  MoveL 9057 to (-391.21, -17.4, -14.38) mm, rotated rx 180 ry 0 rz 0.01 deg; joints [25.24, -41.819, 95.967, -150.014, 58.606, 164.358]
  MoveL 9058 to (-397.59, -19.12, -14.63) mm, rotated rx -180 ry 0 rz 0.01 deg; joints [25.086, -41.563, 95.461, -150.11, 58.344, 164.303]
  MoveL 9059 to (-398.57, -25.65, -14.87) mm, rotated rx 180 ry 0 rz 0.01 deg; joints [24.857, -41.636, 95.647, -150.402, 58.376, 164.507]
  MoveL 9060 to (-392.98, -29.17, -15.11) mm, rotated rx 180 ry 0 rz 0.01 deg; joints [24.827, -41.935, 96.3, -150.543, 58.676, 164.73]
  MoveL 9061 to (-387.52, -25.46, -15.36) mm, rotated rx 180 ry 0 rz 0.01 deg; joints [25.033, -42.088, 96.637, -150.367, 58.894, 164.714]
  MoveL 9062 to (-388.73, -18.96, -15.6) mm, rotated rx 180 ry 0 rz 0.01 deg; joints [25.228, -41.898, 96.253, -150.09, 58.782, 164.486]
  MoveL 9063 to (-395.17, -17.47, -15.85) mm, rotated rx -180 ry 0 rz 0.01 deg; joints [25.178, -41.578, 95.607, -150.047, 58.485, 164.325]
  MoveL 9064 to (-399.11, -22.77, -16.09) mm, rotated rx 180 ry 0 rz 0.01 deg; joints [24.944, -41.498, 95.473, -150.293, 58.37, 164.434]
  MoveL 9065 to (-395.84, -28.51, -16.33) mm, rotated rx 180 ry 0 rz 0.01 deg; joints [24.806, -41.739, 96.011, -150.538, 58.588, 164.688]
  MoveL 9066 to (-389.27, -27.81, -16.58) mm, rotated rx -180 ry 0 rz 0.01 deg; joints [24.93, -41.998, 96.574, -150.49, 58.888, 164.79]
  MoveL 9067 to (-387.28, -21.51, -16.82) mm, rotated rx 180 ry 0 rz 0.01 deg; joints [25.168, -41.951, 96.488, -150.212, 58.922, 164.627]
  MoveL 9068 to (-392.25, -17.16, -17.07) mm, rotated rx -180 ry 0 rz 0.01 deg; joints [25.234, -41.64, 95.854, -150.041, 58.661, 164.4]
  MoveL 9069 to (-398.23, -19.98, -17.31) mm, rotated rx 180 ry 0 rz 0.01 deg; joints [25.05, -41.424, 95.431, -150.184, 58.429, 164.389]
  MoveL 9070 to (-398.04, -26.58, -17.55) mm, rotated rx 180 ry 0 rz 0.01 deg; joints [24.837, -41.548, 95.725, -150.475, 58.515, 164.616]
  MoveL 9071 to (-391.92, -29.05, -17.8) mm, rotated rx -180 ry 0 rz 0.01 deg; joints [24.849, -41.849, 96.383, -150.569, 58.829, 164.814]
  MoveL 9072 to (-387.2, -24.44, -18.04) mm, rotated rx 180 ry 0 rz 0.01 deg; joints [25.073, -41.952, 96.614, -150.355, 59.004, 164.755]
  MoveL 9073 to (-389.54, -18.26, -18.29) mm, rotated rx -180 ry 0 rz 0.01 deg; joints [25.241, -41.72, 96.142, -150.096, 58.844, 164.518]
  MoveL 9074 to (-396.13, -17.93, -18.53) mm, rotated rx 180 ry 0 rz 0.01 deg; joints [25.15, -41.417, 95.53, -150.104, 58.55, 164.392]
  MoveL 9075 to (-399.08, -23.84, -18.77) mm, rotated rx -180 ry 0 rz 0.01 deg; joints [24.912, -41.391, 95.512, -150.374, 58.487, 164.538]
  MoveL 9076 to (-394.85, -28.91, -19.02) mm, rotated rx 180 ry 0 rz 0.01 deg; joints [24.81, -41.661, 96.108, -150.587, 58.742, 164.787]
  MoveL 9077 to (-388.51, -27.06, -19.26) mm, rotated rx 180 ry 0 rz 0.01 deg; joints [24.968, -41.887, 96.602, -150.489, 59.02, 164.848]
  MoveL 9078 to (-387.66, -20.51, -19.51) mm, rotated rx -180 ry 0 rz 0.01 deg; joints [25.197, -41.786, 96.402, -150.204, 59, 164.657]
  MoveL 9079 to (-393.32, -17.11, -19.75) mm, rotated rx -180 ry 0 rz 0.01 deg; joints [25.221, -41.464, 95.746, -150.076, 58.717, 164.448]
  MoveL 9080 to (-398.7, -20.93, -19.99) mm, rotated rx -180 ry 0 rz 0.01 deg; joints [25.013, -41.293, 95.419, -150.262, 58.521, 164.48]
  MoveL 9081 to (-397.36, -27.4, -20.24) mm, rotated rx -180 ry 0 rz 0.01 deg; joints [24.822, -41.464, 95.813, -150.543, 58.66, 164.723]
  MoveL 9082 to (-390.9, -28.76, -20.48) mm, rotated rx -180 ry 0 rz 0.01 deg; joints [24.876, -41.757, 96.454, -150.586, 58.978, 164.891]
  MoveL 9083 to (-387.06, -23.38, -20.73) mm, rotated rx -180 ry 0 rz 0.01 deg; joints [25.112, -41.808, 96.573, -150.343, 59.105, 164.792]
  MoveL 9084 to (-390.45, -17.71, -20.97) mm, rotated rx -180 ry 0 rz 0.01 deg; joints [25.246, -41.541, 96.027, -150.11, 58.901, 164.552]
  MoveL 9085 to (-397, -18.55, -21.21) mm, rotated rx 180 ry 0 rz 0.01 deg; joints [25.118, -41.262, 95.468, -150.168, 58.621, 164.465]
  MoveL 9086 to (-398.86, -24.88, -21.46) mm, rotated rx -180 ry 0 rz 0.01 deg; joints [24.882, -41.292, 95.566, -150.453, 58.612, 164.644]
  MoveL 9087 to (-393.81, -29.13, -21.7) mm, rotated rx -180 ry 0 rz 0.01 deg; joints [24.82, -41.58, 96.202, -150.627, 58.897, 164.881]
  MoveL 9088 to (-387.89, -26.19, -21.95) mm, rotated rx -180 ry 0 rz 0.01 deg; joints [25.007, -41.767, 96.612, -150.483, 59.145, 164.899]
  MoveL 9089 to (-388.21, -19.6, -22.19) mm, rotated rx 180 ry 0 rz 0.01 deg; joints [25.22, -41.615, 96.305, -150.2, 59.07, 164.686]
  MoveL 9090 to (-394.38, -17.24, -22.43) mm, rotated rx -180 ry 0 rz 0.01 deg; joints [25.202, -41.292, 95.646, -150.12, 58.774, 164.502]
  MoveL 9091 to (-399.01, -21.95, -22.68) mm, rotated rx 180 ry 0 rz 0.01 deg; joints [24.977, -41.17, 95.425, -150.341, 58.622, 164.577]
  MoveL 9092 to (-396.54, -28.08, -22.92) mm, rotated rx -180 ry 0 rz 0.01 deg; joints [24.814, -41.383, 95.906, -150.605, 58.809, 164.828]
  MoveL 9093 to (-389.94, -28.28, -23.17) mm, rotated rx 180 ry 0 rz 0.01 deg; joints [24.908, -41.659, 96.51, -150.596, 59.121, 164.961]
  MoveL 9094 to (-387.11, -22.31, -23.41) mm, rotated rx -180 ry 0 rz 0.01 deg; joints [25.148, -41.655, 96.513, -150.33, 59.196, 164.825]
  MoveL 9095 to (-391.45, -17.33, -23.65) mm, rotated rx 180 ry 0 rz 0.01 deg; joints [25.245, -41.361, 95.911, -150.13, 58.956, 164.59]
  MoveL 9096 to (-397.75, -19.31, -23.9) mm, rotated rx 180 ry 0 rz 0.01 deg; joints [25.083, -41.115, 95.422, -150.238, 58.699, 164.544]
  MoveL 9097 to (-398.47, -25.87, -24.14) mm, rotated rx 180 ry 0 rz 0.01 deg; joints [24.858, -41.199, 95.634, -150.529, 58.745, 164.752]
  MoveL 9098 to (-392.74, -29.16, -24.39) mm, rotated rx 180 ry 0 rz 0.01 deg; joints [24.837, -41.497, 96.29, -150.658, 59.051, 164.969]
  MoveL 9099 to (-387.43, -25.23, -24.63) mm, rotated rx -180 ry 0 rz 0.01 deg; joints [25.048, -41.638, 96.603, -150.473, 59.26, 164.944]
  MoveL 9100 to (-388.91, -18.79, -24.88) mm, rotated rx 180 ry 0 rz 0.01 deg; joints [25.237, -41.439, 96.197, -150.201, 59.135, 164.715]
  MoveL 9101 to (-395.4, -17.56, -25.12) mm, rotated rx 180 ry 0 rz 0.01 deg; joints [25.177, -41.124, 95.557, -150.171, 58.835, 164.562]
  MoveL 9102 to (-399.12, -23.01, -25.36) mm, rotated rx -180 ry 0 rz 0.01 deg; joints [24.942, -41.057, 95.449, -150.422, 58.732, 164.677]
  MoveL 9103 to (-395.62, -28.61, -25.61) mm, rotated rx 180 ry 0 rz 0.01 deg; joints [24.812, -41.303, 96.002, -150.659, 58.961, 164.93]
  MoveL 9104 to (-389.09, -27.65, -25.85) mm, rotated rx 180 ry 0 rz 0.01 deg; joints [24.944, -41.554, 96.55, -150.599, 59.259, 165.023]
  MoveL 9105 to (-387.35, -21.27, -26.1) mm, rotated rx 180 ry 0 rz 0.01 deg; joints [25.18, -41.494, 96.438, -150.319, 59.279, 164.855]
  MoveL 9106 to (-392.5, -17.13, -26.34) mm, rotated rx 180 ry 0 rz 0.01 deg; joints [25.237, -41.182, 95.797, -150.159, 59.01, 164.632]
  MoveL 9107 to (-398.35, -20.19, -26.58) mm, rotated rx -180 ry 0 rz 0.01 deg; joints [25.047, -40.977, 95.394, -150.312, 58.784, 164.63]
  MoveL 9108 to (-397.9, -26.78, -26.83) mm, rotated rx -180 ry 0 rz 0.01 deg; joints [24.838, -41.111, 95.713, -150.601, 58.885, 164.859]
  MoveL 9109 to (-391.68, -29, -27.07) mm, rotated rx 180 ry 0 rz 0.01 deg; joints [24.86, -41.409, 96.368, -150.681, 59.202, 165.051]
  MoveL 9110 to (-387.15, -24.2, -27.32) mm, rotated rx -180 ry 0 rz 0.01 deg; joints [25.088, -41.499, 96.574, -150.461, 59.367, 164.984]
  MoveL 9111 to (-389.74, -18.12, -27.56) mm, rotated rx -180 ry 0 rz 0.01 deg; joints [25.248, -41.26, 96.083, -150.208, 59.194, 164.746]
  MoveL 9112 to (-396.34, -18.05, -27.8) mm, rotated rx 180 ry 0 rz 0.01 deg; joints [25.148, -40.963, 95.482, -150.229, 58.901, 164.628]
  MoveL 9113 to (-399.05, -24.08, -28.05) mm, rotated rx 180 ry 0 rz 0.01 deg; joints [24.91, -40.951, 95.49, -150.502, 58.851, 164.781]
  MoveL 9114 to (-394.61, -28.97, -28.29) mm, rotated rx -180 ry 0 rz 0.01 deg; joints [24.817, -41.223, 96.097, -150.704, 59.116, 165.027]
  MoveL 9115 to (-388.35, -26.87, -28.54) mm, rotated rx 180 ry 0 rz 0.01 deg; joints [24.982, -41.439, 96.573, -150.596, 59.389, 165.079]
  MoveL 9116 to (-387.77, -20.29, -28.78) mm, rotated rx -180 ry 0 rz 0.01 deg; joints [25.208, -41.327, 96.348, -150.311, 59.354, 164.884]
  MoveL 9117 to (-393.56, -17.12, -29.02) mm, rotated rx -180 ry 0 rz 0.01 deg; joints [25.222, -41.006, 95.689, -150.195, 59.065, 164.68]
  MoveL 9118 to (-398.79, -21.16, -29.27) mm, rotated rx -180 ry 0 rz 0.01 deg; joints [25.01, -40.847, 95.385, -150.389, 58.878, 164.721]
  MoveL 9119 to (-397.19, -27.57, -29.51) mm, rotated rx 180 ry 0 rz 0.01 deg; joints [24.825, -41.026, 95.8, -150.666, 59.03, 164.965]
  MoveL 9120 to (-390.67, -28.66, -29.76) mm, rotated rx 180 ry 0 rz 0.01 deg; joints [24.888, -41.315, 96.434, -150.696, 59.349, 165.125]
  MoveL 9121 to (-387.06, -23.14, -30) mm, rotated rx -180 ry 0 rz 0.01 deg; joints [25.126, -41.352, 96.526, -150.447, 59.464, 165.019]
  MoveC 9122 to (-392.66, -17.53, -30) mm, rotated rx 180 ry 0 rz 0.01 deg; joints [25.224, -41.005, 95.783, -150.222, 59.148, 164.735] to (-398.27, -23.14, -30) mm, rotated rx -180 ry 0 rz 0.01 deg; joints [24.954, -40.872, 95.512, -150.483, 58.952, 164.813]
  MoveL 9123 to (-398.27, -23.65, -30) mm, rotated rx -180 ry 0 rz 0.01 deg; joints [24.937, -40.881, 95.534, -150.505, 58.957, 164.83]
  MoveC 9124 to (-397.65, -25.14, -30) mm, rotated rx -180 ry 0 rz 0.01 deg; joints [24.898, -40.937, 95.653, -150.568, 59.002, 164.89] to (-396.16, -25.76, -30) mm, rotated rx 180 ry 0 rz 0.01 deg; joints [24.9, -41.013, 95.815, -150.59, 59.077, 164.937]
  MoveL 9125 to (-394.27, -25.76, -30) mm, rotated rx -180 ry 0 rz 0.01 deg; joints [24.929, -41.094, 95.986, -150.585, 59.163, 164.972]
  MoveC 9126 to (-392.51, -24.65, -30) mm, rotated rx -180 ry 0 rz 0.01 deg; joints [24.992, -41.148, 96.099, -150.531, 59.232, 164.969] to (-392.74, -22.58, -30) mm, rotated rx -180 ry 0 rz 0.01 deg; joints [25.057, -41.099, 95.991, -150.442, 59.199, 164.897]
  MoveL 9127 to (-395.33, -19.33, -30) mm, rotated rx -180 ry 0 rz 0.01 deg; joints [25.124, -40.925, 95.618, -150.308, 59.046, 164.744]
  MoveC 9128 to (-397.16, -18.8, -30) mm, rotated rx 180 ry 0 rz 0.01 deg; joints [25.113, -40.836, 95.429, -150.291, 58.956, 164.692] to (-398.27, -20.35, -30) mm, rotated rx -180 ry 0 rz 0.01 deg; joints [25.045, -40.818, 95.395, -150.362, 58.922, 164.723]
  MoveL 9129 to (-398.27, -23.14, -30) mm, rotated rx -180 ry 0 rz 0.01 deg; joints [24.954, -40.872, 95.512, -150.483, 58.952, 164.813]
  MoveL 9130 to (-398.42, -23.66, -30) mm, rotated rx 180 ry 0 rz 0.01 deg; joints [24.935, -40.875, 95.521, -150.506, 58.95, 164.828]
  MoveL 9131 to (-401.46, -28.61, -30) mm, rotated rx 180 ry 0 rz 0.01 deg; joints [24.726, -40.838, 95.452, -150.73, 58.863, 164.932]
  MoveC 9132 to (-402.31, -29.09, -30) mm, rotated rx -180 ry 0 rz 0.01 deg; joints [24.697, -40.81, 95.395, -150.753, 58.829, 164.932] to (-403.17, -28.62, -30) mm, rotated rx 180 ry 0 rz 0.01 deg; joints [24.7, -40.765, 95.297, -150.735, 58.785, 164.901]
  MoveL 9133 to (-403.27, -28.44, -30) mm, rotated rx -180 ry 0 rz 0.01 deg; joints [24.704, -40.757, 95.28, -150.727, 58.778, 164.893]
  MoveL 9134 to (-403.58, -27.62, -30) mm, rotated rx 180 ry 0 rz 0.01 deg; joints [24.726, -40.728, 95.217, -150.693, 58.755, 164.861]
  MoveL 9135 to (-403.78, -26.41, -30) mm, rotated rx 180 ry 0 rz 0.01 deg; joints [24.763, -40.696, 95.149, -150.64, 58.733, 164.818]
  MoveL 9136 to (-403.78, 7.52, -30) mm, rotated rx -180 ry 0 rz 0.01 deg; joints [25.864, -40.028, 93.68, -149.162, 58.365, 163.692]
  MoveL 9137 to (-399.88, -2.51, -30) mm, rotated rx 180 ry 0 rz 0.01 deg; joints [25.601, -40.399, 94.479, -149.59, 58.654, 164.104]
  MoveL 9138 to (-399.67, -2.97, -30) mm, rotated rx -180 ry 0 rz 0.01 deg; joints [25.589, -40.418, 94.519, -149.609, 58.669, 164.123]
  MoveL 9139 to (-395.6, -10.08, -30) mm, rotated rx -180 ry 0 rz 0.01 deg; joints [25.421, -40.734, 95.198, -149.907, 58.933, 164.436]
  MoveL 9140 to (-395.31, -10.51, -30) mm, rotated rx -180 ry 0 rz 0.01 deg; joints [25.412, -40.755, 95.243, -149.925, 58.951, 164.456]
  MoveL 9141 to (-387.56, -20.24, -30) mm, rotated rx -180 ry 0 rz 0.01 deg; joints [25.213, -41.275, 96.359, -150.323, 59.41, 164.917]
  MoveL 9142 to (-387.28, -20.55, -30) mm, rotated rx -180 ry 0 rz 0.01 deg; joints [25.208, -41.293, 96.397, -150.336, 59.426, 164.932]
  MoveL 9143 to (-386.56, -21.26, -30) mm, rotated rx -180 ry 0 rz 0.01 deg; joints [25.196, -41.337, 96.492, -150.364, 59.467, 164.968]
  MoveL 9144 to (-386.09, -21.65, -30) mm, rotated rx -180 ry 0 rz 0.01 deg; joints [25.19, -41.365, 96.551, -150.379, 59.493, 164.989]
  MoveL 9145 to (-377.14, -27.68, -30) mm, rotated rx 180 ry 0 rz 0.01 deg; joints [25.13, -41.858, 97.604, -150.608, 59.963, 165.343]
  MoveL 9146 to (-377.01, -27.76, -30) mm, rotated rx 180 ry 0 rz 0.01 deg; joints [25.129, -41.865, 97.619, -150.611, 59.97, 165.348]
  MoveL 9147 to (-375.25, -28.84, -30) mm, rotated rx 180 ry 0 rz 0.01 deg; joints [25.121, -41.96, 97.821, -150.65, 60.061, 165.413]
  MoveL 9148 to (-374.65, -29.13, -30) mm, rotated rx -180 ry 0 rz 0.01 deg; joints [25.12, -41.99, 97.886, -150.66, 60.091, 165.433]
  MoveL 9149 to (-373.52, -29.55, -30) mm, rotated rx -180 ry 0 rz 0.01 deg; joints [25.124, -42.046, 98.004, -150.674, 60.147, 165.466]
  MoveL 9150 to (-373.3, -29.62, -30) mm, rotated rx -180 ry 0 rz 0.01 deg; joints [25.125, -42.056, 98.027, -150.676, 60.158, 165.472]
  MoveL 9151 to (-367.68, -31.27, -30) mm, rotated rx 180 ry 0 rz 0.01 deg; joints [25.158, -42.322, 98.592, -150.723, 60.428, 165.623]
  MoveL 9152 to (-398.96, -31.27, -30) mm, rotated rx 180 ry 0 rz 0.01 deg; joints [24.677, -40.996, 95.791, -150.838, 59.007, 165.064]
  MoveL 9153 to (-399.88, -31.14, -30) mm, rotated rx 180 ry 0 rz 0.01 deg; joints [24.667, -40.954, 95.701, -150.835, 58.963, 165.043]
  MoveL 9154 to (-400.74, -30.86, -30) mm, rotated rx 180 ry 0 rz 0.01 deg; joints [24.663, -40.912, 95.612, -150.826, 58.921, 165.018]
  MoveL 9155 to (-401.19, -30.62, -30) mm, rotated rx -180 ry 0 rz 0.01 deg; joints [24.664, -40.888, 95.561, -150.816, 58.898, 165.002]
  MoveL 9156 to (-401.26, -29.55, -30) mm, rotated rx 180 ry 0 rz 0.01 deg; joints [24.698, -40.865, 95.51, -150.77, 58.883, 164.966]
  MoveL 9157 to (-398.54, -27.51, -30) mm, rotated rx -180 ry 0 rz 0.01 deg; joints [24.806, -40.943, 95.672, -150.674, 58.986, 164.95]
  MoveL 9158 to (-393.94, -23.88, -30) mm, rotated rx 180 ry 0 rz 0.01 deg; joints [24.996, -41.072, 95.937, -150.502, 59.158, 164.917]
  MoveL 9159 to (-392.18, -23.29, -30) mm, rotated rx -180 ry 0 rz 0.01 deg; joints [25.042, -41.136, 96.071, -150.471, 59.232, 164.93]
  MoveL 9160 to (-391.94, -22.8, -30) mm, rotated rx 180 ry 0 rz 0.01 deg; joints [25.062, -41.137, 96.072, -150.449, 59.238, 164.919]
  MoveL 9161 to (-397.13, -18.72, -30.24) mm, rotated rx 180 ry 0 rz 0.01 deg; joints [25.116, -40.824, 95.428, -150.29, 58.966, 164.697]
  MoveL 9162 to (-402.95, -21.84, -30.49) mm, rotated rx 180 ry 0 rz 0.01 deg; joints [24.926, -40.621, 95.029, -150.445, 58.741, 164.696]
  MoveL 9163 to (-402.43, -28.42, -30.73) mm, rotated rx 180 ry 0 rz 0.01 deg; joints [24.718, -40.757, 95.353, -150.733, 58.845, 164.926]
  MoveL 9164 to (-396.2, -30.59, -30.98) mm, rotated rx 180 ry 0 rz 0.01 deg; joints [24.742, -41.055, 96.009, -150.812, 59.165, 165.117]
  MoveL 9165 to (-391.71, -25.75, -31.22) mm, rotated rx -180 ry 0 rz 0.01 deg; joints [24.969, -41.144, 96.212, -150.591, 59.328, 165.049]
  MoveL 9166 to (-394.34, -19.69, -31.46) mm, rotated rx -180 ry 0 rz 0.01 deg; joints [25.128, -40.904, 95.717, -150.339, 59.151, 164.811]
  MoveL 9167 to (-400.94, -19.67, -31.71) mm, rotated rx -180 ry 0 rz 0.01 deg; joints [25.028, -40.607, 95.115, -150.361, 58.857, 164.693]
  MoveL 9168 to (-403.61, -25.71, -31.95) mm, rotated rx 180 ry 0 rz 0.01 deg; joints [24.79, -40.596, 95.126, -150.633, 58.808, 164.846]
  MoveL 9169 to (-399.15, -30.58, -32.2) mm, rotated rx -180 ry 0 rz 0.01 deg; joints [24.698, -40.869, 95.735, -150.836, 59.076, 165.093]
  MoveL 9170 to (-392.9, -28.44, -32.44) mm, rotated rx -180 ry 0 rz 0.01 deg; joints [24.863, -41.085, 96.212, -150.727, 59.35, 165.144]
  MoveL 9171 to (-392.35, -21.87, -32.68) mm, rotated rx 180 ry 0 rz 0.01 deg; joints [25.088, -40.971, 95.984, -150.442, 59.313, 164.949]
  MoveL 9172 to (-398.15, -18.72, -32.93) mm, rotated rx -180 ry 0 rz 0.01 deg; joints [25.102, -40.65, 95.323, -150.326, 59.022, 164.745]
  MoveL 9173 to (-403.36, -22.77, -33.17) mm, rotated rx -180 ry 0 rz 0.01 deg; joints [24.891, -40.491, 95.019, -150.52, 58.835, 164.785]
  MoveL 9174 to (-401.74, -29.17, -33.41) mm, rotated rx 180 ry 0 rz 0.01 deg; joints [24.706, -40.671, 95.435, -150.797, 58.988, 165.029]
  MoveL 9175 to (-395.23, -30.26, -33.66) mm, rotated rx -180 ry 0 rz 0.01 deg; joints [24.769, -40.96, 96.071, -150.827, 59.309, 165.19]
  MoveL 9176 to (-391.62, -24.73, -33.9) mm, rotated rx 180 ry 0 rz 0.01 deg; joints [25.006, -40.997, 96.165, -150.579, 59.424, 165.084]
  MoveL 9177 to (-395.24, -19.21, -34.15) mm, rotated rx 180 ry 0 rz 0.01 deg; joints [25.132, -40.725, 95.603, -150.354, 59.208, 164.845]
  MoveL 9178 to (-401.75, -20.3, -34.39) mm, rotated rx 180 ry 0 rz 0.01 deg; joints [24.997, -40.455, 95.056, -150.423, 58.929, 164.765]
  MoveL 9179 to (-403.36, -26.7, -34.63) mm, rotated rx -180 ry 0 rz 0.01 deg; joints [24.763, -40.496, 95.178, -150.709, 58.934, 164.95]
  MoveL 9180 to (-398.14, -30.74, -34.88) mm, rotated rx -180 ry 0 rz 0.01 deg; joints [24.709, -40.785, 95.822, -150.872, 59.228, 165.183]
  MoveL 9181 to (-392.34, -27.59, -35.12) mm, rotated rx -180 ry 0 rz 0.01 deg; joints [24.901, -40.961, 96.214, -150.72, 59.47, 165.193]
  MoveL 9182 to (-392.91, -21.01, -35.37) mm, rotated rx -180 ry 0 rz 0.01 deg; joints [25.109, -40.8, 95.885, -150.44, 59.382, 164.978]
  MoveL 9183 to (-399.15, -18.89, -35.61) mm, rotated rx -180 ry 0 rz 0.01 deg; joints [25.083, -40.48, 95.226, -150.37, 59.08, 164.798]
  MoveL 9184 to (-403.61, -23.76, -35.85) mm, rotated rx -180 ry 0 rz 0.01 deg; joints [24.856, -40.37, 95.025, -150.597, 58.937, 164.879]
  MoveL 9185 to (-400.93, -29.8, -36.1) mm, rotated rx -180 ry 0 rz 0.01 deg; joints [24.699, -40.587, 95.522, -150.854, 59.136, 165.13]
  MoveL 9186 to (-394.33, -29.77, -36.34) mm, rotated rx -180 ry 0 rz 0.01 deg; joints [24.8, -40.858, 96.119, -150.836, 59.449, 165.257]
  MoveL 9187 to (-391.71, -23.71, -36.59) mm, rotated rx -180 ry 0 rz 0.01 deg; joints [25.04, -40.843, 96.101, -150.568, 59.513, 165.117]
  MoveL 9188 to (-396.2, -18.88, -36.83) mm, rotated rx -180 ry 0 rz 0.01 deg; joints [25.129, -40.547, 95.488, -150.375, 59.263, 164.883]
  MoveL 9189 to (-402.44, -21.05, -37.07) mm, rotated rx 180 ry 0 rz 0.01 deg; joints [24.963, -40.309, 95.012, -150.491, 59.008, 164.843]
  MoveL 9190 to (-402.94, -27.63, -37.32) mm, rotated rx -180 ry 0 rz 0.01 deg; joints [24.74, -40.401, 95.242, -150.781, 59.066, 165.053]
  MoveL 9191 to (-397.12, -30.74, -37.56) mm, rotated rx -180 ry 0 rz 0.01 deg; joints [24.727, -40.697, 95.901, -150.901, 59.379, 165.267]
  MoveL 9192 to (-391.94, -26.65, -37.8) mm, rotated rx 180 ry 0 rz 0.01 deg; joints [24.94, -40.83, 96.198, -150.71, 59.582, 165.237]
  MoveL 9193 to (-393.6, -20.26, -38.05) mm, rotated rx -180 ry 0 rz 0.01 deg; joints [25.125, -40.626, 95.777, -150.442, 59.444, 165.007]
  MoveL 9194 to (-400.12, -19.23, -38.29) mm, rotated rx 180 ry 0 rz 0.01 deg; joints [25.059, -40.315, 95.14, -150.42, 59.142, 164.858]
  MoveL 9195 to (-403.69, -24.78, -38.54) mm, rotated rx -180 ry 0 rz 0.01 deg; joints [24.823, -40.255, 95.048, -150.674, 59.047, 164.977]
  MoveL 9196 to (-400.03, -30.28, -38.78) mm, rotated rx 180 ry 0 rz 0.01 deg; joints [24.699, -40.504, 95.611, -150.904, 59.286, 165.228]
  MoveL 9197 to (-393.53, -29.14, -39.02) mm, rotated rx -180 ry 0 rz 0.01 deg; joints [24.835, -40.749, 96.152, -150.838, 59.583, 165.317]
  MoveL 9198 to (-391.97, -22.72, -39.27) mm, rotated rx -180 ry 0 rz 0.01 deg; joints [25.07, -40.682, 96.023, -150.558, 59.593, 165.147]
  MoveL 9199 to (-397.21, -18.72, -39.51) mm, rotated rx -180 ry 0 rz 0.01 deg; joints [25.121, -40.37, 95.376, -150.404, 59.317, 164.926]
  MoveL 9200 to (-402.99, -21.91, -39.76) mm, rotated rx 180 ry 0 rz 0.01 deg; joints [24.928, -40.172, 94.985, -150.562, 59.094, 164.927]
  MoveL 9201 to (-402.38, -28.48, -40) mm, rotated rx 180 ry 0 rz 0.01 deg; joints [24.723, -40.311, 95.316, -150.848, 59.204, 165.157]
  MoveC 9202 to (-394.5, -29.39, -40) mm, rotated rx 180 ry 0 rz 0.01 deg; joints [24.812, -40.664, 96.07, -150.863, 59.578, 165.331] to (-393.6, -21.51, -40) mm, rotated rx 180 ry 0 rz 0.01 deg; joints [25.085, -40.554, 95.82, -150.52, 59.533, 165.095]
  MoveL 9203 to (-395.33, -19.33, -40) mm, rotated rx 180 ry 0 rz 0.01 deg; joints [25.13, -40.438, 95.571, -150.431, 59.429, 164.993]
  MoveC 9204 to (-397.17, -18.8, -40) mm, rotated rx -180 ry 0 rz 0.01 deg; joints [25.119, -40.35, 95.382, -150.413, 59.338, 164.941] to (-398.27, -20.35, -40) mm, rotated rx 180 ry 0 rz 0.01 deg; joints [25.051, -40.332, 95.347, -150.484, 59.305, 164.971]
  MoveL 9205 to (-398.27, -23.65, -40) mm, rotated rx -180 ry 0 rz 0.01 deg; joints [24.943, -40.395, 95.486, -150.627, 59.341, 165.077]
  MoveC 9206 to (-397.65, -25.14, -40) mm, rotated rx 180 ry 0 rz 0.01 deg; joints [24.904, -40.45, 95.606, -150.69, 59.386, 165.137] to (-396.16, -25.76, -40) mm, rotated rx 180 ry 0 rz 0.01 deg; joints [24.906, -40.525, 95.767, -150.712, 59.462, 165.185]
  MoveL 9207 to (-394.28, -25.76, -40) mm, rotated rx -180 ry 0 rz 0.01 deg; joints [24.935, -40.605, 95.938, -150.706, 59.549, 165.219]
  MoveC 9208 to (-392.51, -24.65, -40) mm, rotated rx -180 ry 0 rz 0.01 deg; joints [24.998, -40.66, 96.051, -150.652, 59.618, 165.216] to (-392.75, -22.58, -40) mm, rotated rx 180 ry 0 rz 0.01 deg; joints [25.063, -40.611, 95.943, -150.563, 59.584, 165.146]
  MoveL 9209 to (-393.6, -21.51, -40) mm, rotated rx 180 ry 0 rz 0.01 deg; joints [25.085, -40.554, 95.82, -150.52, 59.533, 165.095]
  MoveL 9210 to (-394.1, -21.13, -39.83) mm, rotated rx -180 ry 0 rz 0.01 deg; joints [25.09, -40.534, 95.76, -150.503, 59.499, 165.07]
  MoveL 9211 to (-394.55, -21.03, -39.37) mm, rotated rx 180 ry 0 rz 0.01 deg; joints [25.086, -40.535, 95.717, -150.494, 59.46, 165.047]
  MoveL 9212 to (-394.72, -21.04, -38.73) mm, rotated rx 180 ry 0 rz 0.01 deg; joints [25.083, -40.559, 95.705, -150.487, 59.427, 165.028]
  Set speed (1000.0 mm/s)
  MoveL 9213 to (-394.72, -21.04, 11) mm, rotated rx 180 ry 0 rz 0.01 deg; joints [25.051, -42.942, 95.855, -149.84, 57.481, 163.743]
  Set speed (1000.0 mm/s)
  MoveL 9214 to (-396.98, -23.89, 11) mm, rotated rx -180 ry 0 rz 0.01 deg; joints [24.923, -42.898, 95.771, -149.972, 57.408, 163.798]
  Set speed (100.0 mm/s)
  MoveL 9215 to (-396.98, -23.89, -19) mm, rotated rx -180 ry 0 rz 0.01 deg; joints [24.942, -41.473, 95.704, -150.373, 58.592, 164.584]
  MoveL 9216 to (-396.98, -23.89, -38.73) mm, rotated rx 180 ry 0 rz 0.01 deg; joints [24.954, -40.517, 95.621, -150.618, 59.355, 165.078]
  MoveL 9217 to (-398.09, -24.52, -40) mm, rotated rx -180 ry 0 rz 0.01 deg; joints [24.918, -40.419, 95.54, -150.664, 59.359, 165.109]
  MoveL 9218 to (-403.58, -27.62, -40) mm, rotated rx -180 ry 0 rz 0.01 deg; joints [24.733, -40.242, 95.17, -150.814, 59.139, 165.107]
  MoveL 9219 to (-403.78, -26.41, -40) mm, rotated rx -180 ry 0 rz 0.01 deg; joints [24.769, -40.211, 95.101, -150.762, 59.116, 165.064]
  MoveL 9220 to (-403.78, 7.52, -40) mm, rotated rx -180 ry 0 rz 0.01 deg; joints [25.87, -39.549, 93.633, -149.29, 58.738, 163.947]
  MoveL 9221 to (-399.88, -2.51, -40) mm, rotated rx 180 ry 0 rz 0.01 deg; joints [25.607, -39.917, 94.432, -149.716, 59.031, 164.357]
  MoveL 9222 to (-399.67, -2.97, -40) mm, rotated rx -180 ry 0 rz 0.01 deg; joints [25.596, -39.935, 94.472, -149.735, 59.046, 164.377]
  MoveL 9223 to (-395.6, -10.08, -40) mm, rotated rx -180 ry 0 rz 0.01 deg; joints [25.428, -40.249, 95.151, -150.031, 59.314, 164.688]
  MoveL 9224 to (-395.31, -10.51, -40) mm, rotated rx 180 ry 0 rz 0.01 deg; joints [25.418, -40.27, 95.196, -150.049, 59.332, 164.707]
  MoveL 9225 to (-387.58, -20.24, -40) mm, rotated rx -180 ry 0 rz 0.01 deg; joints [25.22, -40.785, 96.31, -150.444, 59.795, 165.166]
  MoveL 9226 to (-387.28, -20.57, -40) mm, rotated rx -180 ry 0 rz 0.01 deg; joints [25.213, -40.804, 96.351, -150.458, 59.813, 165.182]
  MoveL 9227 to (-386.54, -21.28, -40) mm, rotated rx 180 ry 0 rz 0.01 deg; joints [25.201, -40.849, 96.447, -150.486, 59.854, 165.218]
  MoveL 9228 to (-386.09, -21.64, -40) mm, rotated rx 180 ry 0 rz 0.01 deg; joints [25.196, -40.875, 96.503, -150.5, 59.879, 165.238]
  MoveL 9229 to (-376.26, -28.29, -40) mm, rotated rx -180 ry 0 rz 0.01 deg; joints [25.129, -41.412, 97.661, -150.749, 60.401, 165.627]
  MoveL 9230 to (-375.91, -28.5, -40) mm, rotated rx 180 ry 0 rz 0.01 deg; joints [25.128, -41.431, 97.701, -150.756, 60.419, 165.639]
  MoveL 9231 to (-374.74, -29.1, -40) mm, rotated rx 180 ry 0 rz 0.01 deg; joints [25.126, -41.491, 97.829, -150.777, 60.479, 165.679]
  MoveL 9232 to (-374.21, -29.32, -40) mm, rotated rx -180 ry 0 rz 0.01 deg; joints [25.127, -41.517, 97.886, -150.785, 60.506, 165.695]
  MoveL 9233 to (-370.46, -30.49, -40) mm, rotated rx 180 ry 0 rz 0.01 deg; joints [25.147, -41.695, 98.268, -150.819, 60.689, 165.799]
  MoveL 9234 to (-370.4, -30.51, -40) mm, rotated rx -180 ry 0 rz 0.01 deg; joints [25.147, -41.697, 98.273, -150.82, 60.692, 165.8]
  MoveL 9235 to (-367.83, -31.27, -40) mm, rotated rx 180 ry 0 rz 0.01 deg; joints [25.162, -41.818, 98.531, -150.841, 60.816, 165.869]
  MoveL 9236 to (-398.96, -31.27, -40) mm, rotated rx 180 ry 0 rz 0.01 deg; joints [24.683, -40.509, 95.743, -150.959, 59.393, 165.309]
  MoveL 9237 to (-399.88, -31.14, -40) mm, rotated rx 180 ry 0 rz 0.01 deg; joints [24.673, -40.467, 95.654, -150.956, 59.349, 165.288]
  MoveL 9238 to (-400.74, -30.86, -40) mm, rotated rx -180 ry 0 rz 0.01 deg; joints [24.669, -40.425, 95.565, -150.946, 59.306, 165.264]
  MoveL 9239 to (-401.19, -30.62, -40) mm, rotated rx 180 ry 0 rz 0.01 deg; joints [24.671, -40.402, 95.514, -150.937, 59.283, 165.247]
  MoveL 9240 to (-401.09, -28.82, -40) mm, rotated rx -180 ry 0 rz 0.01 deg; joints [24.731, -40.372, 95.448, -150.859, 59.268, 165.192]
  MoveL 9241 to (-392.1, -25.03, -40) mm, rotated rx 180 ry 0 rz 0.01 deg; joints [24.992, -40.684, 96.104, -150.667, 59.641, 165.236]
  MoveL 9242 to (-389.72, -19.06, -40.24) mm, rotated rx 180 ry 0 rz 0.01 deg; joints [25.225, -40.66, 96.066, -150.404, 59.693, 165.094]
  MoveL 9243 to (-394.08, -14.33, -40.47) mm, rotated rx 180 ry 0 rz 0.01 deg; joints [25.313, -40.373, 95.469, -150.216, 59.449, 164.866]
  MoveL 9244 to (-400.23, -16.22, -40.71) mm, rotated rx -180 ry 0 rz 0.01 deg; joints [25.157, -40.135, 94.989, -150.319, 59.195, 164.818]
  MoveL 9245 to (-401.17, -22.59, -40.95) mm, rotated rx -180 ry 0 rz 0.01 deg; joints [24.935, -40.204, 95.172, -150.601, 59.231, 165.012]
  MoveL 9246 to (-395.85, -26.19, -41.18) mm, rotated rx 180 ry 0 rz 0.01 deg; joints [24.898, -40.489, 95.808, -150.743, 59.526, 165.233]
  MoveL 9247 to (-390.3, -22.93, -41.42) mm, rotated rx 180 ry 0 rz 0.01 deg; joints [25.09, -40.651, 96.171, -150.587, 59.755, 165.237]
  MoveL 9248 to (-390.84, -16.53, -41.66) mm, rotated rx 180 ry 0 rz 0.01 deg; joints [25.292, -40.495, 95.85, -150.315, 59.668, 165.027]
  MoveL 9249 to (-396.85, -14.24, -41.89) mm, rotated rx -180 ry 0 rz 0.01 deg; joints [25.274, -40.184, 95.206, -150.238, 59.374, 164.847]
  MoveL 9250 to (-401.5, -18.68, -42.13) mm, rotated rx 180 ry 0 rz 0.01 deg; joints [25.058, -40.058, 94.971, -150.447, 59.217, 164.908]
  MoveL 9251 to (-399.51, -24.79, -42.37) mm, rotated rx -180 ry 0 rz 0.01 deg; joints [24.889, -40.248, 95.41, -150.708, 59.387, 165.149]
  MoveL 9252 to (-393.14, -25.64, -42.61) mm, rotated rx 180 ry 0 rz 0.01 deg; joints [24.958, -40.524, 96.023, -150.728, 59.7, 165.3]
  MoveL 9253 to (-389.62, -20.25, -42.84) mm, rotated rx -180 ry 0 rz 0.01 deg; joints [25.189, -40.56, 96.112, -150.486, 59.811, 165.199]
  MoveL 9254 to (-392.96, -14.76, -43.08) mm, rotated rx -180 ry 0 rz 0.01 deg; joints [25.318, -40.301, 95.575, -150.263, 59.605, 164.966]
  MoveL 9255 to (-399.36, -15.4, -43.32) mm, rotated rx 180 ry 0 rz 0.01 deg; joints [25.199, -40.029, 95.019, -150.313, 59.325, 164.872]
  MoveL 9256 to (-401.55, -21.44, -43.55) mm, rotated rx -180 ry 0 rz 0.01 deg; joints [24.968, -40.04, 95.076, -150.583, 59.3, 165.032]
  MoveL 9257 to (-397.04, -26.03, -43.79) mm, rotated rx 180 ry 0 rz 0.01 deg; joints [24.887, -40.307, 95.679, -150.771, 59.569, 165.269]
  MoveL 9258 to (-390.95, -23.94, -44.03) mm, rotated rx -180 ry 0 rz 0.01 deg; joints [25.048, -40.515, 96.141, -150.664, 59.836, 165.321]
  MoveL 9259 to (-390.21, -17.55, -44.26) mm, rotated rx 180 ry 0 rz 0.01 deg; joints [25.27, -40.413, 95.936, -150.388, 59.808, 165.136]
  MoveL 9260 to (-395.65, -14.12, -44.5) mm, rotated rx -180 ry 0 rz 0.01 deg; joints [25.298, -40.105, 95.296, -150.261, 59.527, 164.93]
  MoveC 9261 to (-401.47, -19.94, -44.5) mm, rotated rx 180 ry 0 rz 0.01 deg; joints [25.019, -39.968, 95.014, -150.53, 59.323, 165.008] to (-395.65, -25.76, -44.5) mm, rotated rx -180 ry 0 rz 0.01 deg; joints [24.917, -40.326, 95.789, -150.763, 59.658, 165.304]
  MoveL 9262 to (-394.28, -25.76, -44.5) mm, rotated rx -180 ry 0 rz 0.01 deg; joints [24.938, -40.385, 95.914, -150.759, 59.721, 165.329]
  MoveC 9263 to (-392.52, -24.66, -44.5) mm, rotated rx 180 ry 0 rz 0.01 deg; joints [25.001, -40.439, 96.027, -150.705, 59.79, 165.326] to (-392.75, -22.59, -44.5) mm, rotated rx -180 ry 0 rz 0.01 deg; joints [25.066, -40.39, 95.919, -150.617, 59.756, 165.256]
  MoveL 9264 to (-395.33, -19.33, -44.5) mm, rotated rx 180 ry 0 rz 0.01 deg; joints [25.133, -40.218, 95.547, -150.485, 59.6, 165.103]
  MoveC 9265 to (-397.17, -18.8, -44.5) mm, rotated rx 180 ry 0 rz 0.01 deg; joints [25.122, -40.13, 95.358, -150.467, 59.509, 165.052] to (-398.27, -20.35, -44.5) mm, rotated rx 180 ry 0 rz 0.01 deg; joints [25.054, -40.113, 95.323, -150.538, 59.476, 165.081]
  MoveL 9266 to (-398.27, -23.65, -44.5) mm, rotated rx 180 ry 0 rz 0.01 deg; joints [24.946, -40.175, 95.462, -150.68, 59.513, 165.187]
  MoveC 9267 to (-397.65, -25.14, -44.5) mm, rotated rx 180 ry 0 rz 0.01 deg; joints [24.907, -40.23, 95.582, -150.743, 59.558, 165.247] to (-396.16, -25.76, -44.5) mm, rotated rx 180 ry 0 rz 0.01 deg; joints [24.909, -40.305, 95.744, -150.765, 59.634, 165.294]
  MoveL 9268 to (-395.65, -25.76, -44.5) mm, rotated rx 180 ry 0 rz 0.01 deg; joints [24.917, -40.326, 95.789, -150.763, 59.658, 165.304]
  MoveL 9269 to (-395.47, -27.75, -44.5) mm, rotated rx 180 ry 0 rz 0.01 deg; joints [24.854, -40.371, 95.889, -150.849, 59.688, 165.371]
  MoveL 9270 to (-400.89, -28.76, -44.5) mm, rotated rx -180 ry 0 rz 0.01 deg; joints [24.739, -40.16, 95.439, -150.909, 59.448, 165.303]
  MoveL 9271 to (-401.19, -30.62, -44.5) mm, rotated rx -180 ry 0 rz 0.01 deg; joints [24.674, -40.182, 95.49, -150.99, 59.455, 165.356]
  MoveL 9272 to (-400.74, -30.86, -44.5) mm, rotated rx -180 ry 0 rz 0.01 deg; joints [24.672, -40.205, 95.541, -151, 59.478, 165.373]
  MoveL 9273 to (-399.88, -31.14, -44.5) mm, rotated rx -180 ry 0 rz 0.01 deg; joints [24.676, -40.247, 95.63, -151.009, 59.521, 165.397]
  MoveL 9274 to (-398.96, -31.27, -44.5) mm, rotated rx -180 ry 0 rz 0.01 deg; joints [24.686, -40.289, 95.719, -151.012, 59.566, 165.418]
  MoveL 9275 to (-367.79, -31.27, -44.5) mm, rotated rx 180 ry 0 rz 0.01 deg; joints [25.165, -41.594, 98.511, -150.892, 60.994, 165.98]
  MoveL 9276 to (-373.89, -29.44, -44.5) mm, rotated rx 180 ry 0 rz 0.01 deg; joints [25.131, -41.309, 97.896, -150.84, 60.697, 165.816]
  MoveL 9277 to (-374.38, -29.25, -44.5) mm, rotated rx -180 ry 0 rz 0.01 deg; joints [25.13, -41.285, 97.844, -150.834, 60.673, 165.801]
  MoveL 9278 to (-375.83, -28.55, -44.5) mm, rotated rx 180 ry 0 rz 0.01 deg; joints [25.13, -41.211, 97.686, -150.81, 60.599, 165.753]
  MoveL 9279 to (-376.26, -28.3, -44.5) mm, rotated rx -180 ry 0 rz 0.01 deg; joints [25.132, -41.189, 97.637, -150.801, 60.576, 165.737]
  MoveL 9280 to (-386.1, -21.64, -44.5) mm, rotated rx 180 ry 0 rz 0.01 deg; joints [25.199, -40.653, 96.478, -150.553, 60.052, 165.349]
  MoveL 9281 to (-386.54, -21.28, -44.5) mm, rotated rx 180 ry 0 rz 0.01 deg; joints [25.204, -40.628, 96.424, -150.539, 60.028, 165.329]
  MoveL 9282 to (-387.27, -20.58, -44.5) mm, rotated rx 180 ry 0 rz 0.01 deg; joints [25.216, -40.583, 96.328, -150.511, 59.986, 165.293]
  MoveL 9283 to (-387.59, -20.24, -44.5) mm, rotated rx 180 ry 0 rz 0.01 deg; joints [25.222, -40.564, 96.285, -150.498, 59.968, 165.277]
  MoveL 9284 to (-395.31, -10.51, -44.5) mm, rotated rx 180 ry 0 rz 0.01 deg; joints [25.421, -40.05, 95.172, -150.103, 59.502, 164.819]
  MoveL 9285 to (-395.6, -10.08, -44.5) mm, rotated rx 180 ry 0 rz 0.01 deg; joints [25.43, -40.03, 95.127, -150.086, 59.484, 164.8]
  MoveL 9286 to (-399.67, -2.97, -44.5) mm, rotated rx -180 ry 0 rz 0.01 deg; joints [25.598, -39.717, 94.448, -149.79, 59.215, 164.489]
  MoveL 9287 to (-399.88, -2.52, -44.5) mm, rotated rx 180 ry 0 rz 0.01 deg; joints [25.609, -39.699, 94.409, -149.771, 59.2, 164.47]
  MoveL 9288 to (-403.78, 7.44, -44.5) mm, rotated rx -180 ry 0 rz 0.01 deg; joints [25.87, -39.334, 93.613, -149.35, 58.906, 164.064]
  MoveL 9289 to (-403.78, -26.41, -44.5) mm, rotated rx 180 ry 0 rz 0.01 deg; joints [24.772, -39.992, 95.077, -150.816, 59.288, 165.173]
  MoveL 9290 to (-403.58, -27.62, -44.5) mm, rotated rx -180 ry 0 rz 0.01 deg; joints [24.735, -40.023, 95.146, -150.868, 59.31, 165.216]
  MoveL 9291 to (-403.27, -28.44, -44.5) mm, rotated rx 180 ry 0 rz 0.01 deg; joints [24.713, -40.052, 95.208, -150.903, 59.334, 165.248]
  MoveL 9292 to (-403.17, -28.62, -44.5) mm, rotated rx -180 ry 0 rz 0.01 deg; joints [24.709, -40.06, 95.226, -150.91, 59.341, 165.256]
  MoveL 9293 to (-402.57, -28.71, -44.5) mm, rotated rx 180 ry 0 rz 0.01 deg; joints [24.715, -40.087, 95.284, -150.912, 59.369, 165.27]
  MoveL 9294 to (-401.12, -27.44, -44.5) mm, rotated rx 180 ry 0 rz 0.01 deg; joints [24.779, -40.125, 95.363, -150.853, 59.423, 165.256]
  MoveL 9295 to (-394.75, -24.03, -44.5) mm, rotated rx -180 ry 0 rz 0.01 deg; joints [24.988, -40.332, 95.798, -150.686, 59.68, 165.265]
  MoveL 9296 to (-392.32, -23.48, -44.5) mm, rotated rx 180 ry 0 rz 0.01 deg; joints [25.043, -40.425, 95.995, -150.654, 59.786, 165.292]
  MoveL 9297 to (-391.94, -22.81, -44.5) mm, rotated rx -180 ry 0 rz 0.01 deg; joints [25.07, -40.428, 96.001, -150.624, 59.796, 165.278]
  MoveL 9298 to (-397.13, -18.73, -44.74) mm, rotated rx 180 ry 0 rz 0.01 deg; joints [25.125, -40.119, 95.357, -150.467, 59.52, 165.056]
  MoveL 9299 to (-402.95, -21.83, -44.99) mm, rotated rx 180 ry 0 rz 0.01 deg; joints [24.935, -39.917, 94.957, -150.621, 59.294, 165.053]
  MoveL 9300 to (-402.44, -28.41, -45.23) mm, rotated rx -180 ry 0 rz 0.01 deg; joints [24.727, -40.051, 95.279, -150.907, 59.4, 165.28]
  MoveL 9301 to (-396.21, -30.59, -45.48) mm, rotated rx -180 ry 0 rz 0.01 deg; joints [24.75, -40.345, 95.936, -150.985, 59.723, 165.471]
  MoveL 9302 to (-391.72, -25.76, -45.72) mm, rotated rx 180 ry 0 rz 0.01 deg; joints [24.978, -40.433, 96.139, -150.764, 59.886, 165.406]
  MoveL 9303 to (-394.34, -19.7, -45.96) mm, rotated rx -180 ry 0 rz 0.01 deg; joints [25.137, -40.196, 95.644, -150.515, 59.706, 165.17]
  MoveL 9304 to (-400.94, -19.67, -46.21) mm, rotated rx 180 ry 0 rz 0.01 deg; joints [25.037, -39.902, 95.042, -150.537, 59.409, 165.051]
  MoveL 9305 to (-403.62, -25.71, -46.45) mm, rotated rx -180 ry 0 rz 0.01 deg; joints [24.799, -39.89, 95.051, -150.808, 59.361, 165.201]
  MoveL 9306 to (-399.16, -30.58, -46.7) mm, rotated rx -180 ry 0 rz 0.01 deg; joints [24.707, -40.16, 95.66, -151.008, 59.633, 165.446]
  MoveL 9307 to (-392.91, -28.45, -46.94) mm, rotated rx 180 ry 0 rz 0.01 deg; joints [24.872, -40.373, 96.137, -150.899, 59.908, 165.499]
  MoveL 9308 to (-392.35, -21.88, -47.18) mm, rotated rx 180 ry 0 rz 0.01 deg; joints [25.097, -40.261, 95.91, -150.616, 59.869, 165.306]
  MoveL 9309 to (-398.15, -18.72, -47.43) mm, rotated rx 180 ry 0 rz 0.01 deg; joints [25.111, -39.944, 95.249, -150.502, 59.574, 165.103]
  MoveL 9310 to (-403.36, -22.77, -47.67) mm, rotated rx 180 ry 0 rz 0.01 deg; joints [24.9, -39.786, 94.943, -150.695, 59.386, 165.14]
  MoveL 9311 to (-401.75, -29.17, -47.91) mm, rotated rx 180 ry 0 rz 0.01 deg; joints [24.715, -39.963, 95.358, -150.969, 59.543, 165.382]
  MoveL 9312 to (-395.24, -30.26, -48.16) mm, rotated rx -180 ry 0 rz 0.01 deg; joints [24.777, -40.248, 95.994, -150.999, 59.867, 165.543]
  MoveL 9313 to (-391.63, -24.74, -48.4) mm, rotated rx -180 ry 0 rz 0.01 deg; joints [25.015, -40.285, 96.088, -150.751, 59.981, 165.44]
  MoveL 9314 to (-395.24, -19.21, -48.65) mm, rotated rx -180 ry 0 rz 0.01 deg; joints [25.141, -40.017, 95.527, -150.528, 59.761, 165.203]
  MoveL 9315 to (-401.75, -20.3, -48.89) mm, rotated rx 180 ry 0 rz 0.01 deg; joints [25.006, -39.748, 94.979, -150.598, 59.48, 165.121]
  MoveL 9316 to (-403.37, -26.7, -49.13) mm, rotated rx 180 ry 0 rz 0.01 deg; joints [24.772, -39.788, 95.1, -150.882, 59.486, 165.302]
  MoveL 9317 to (-398.15, -30.75, -49.38) mm, rotated rx 180 ry 0 rz 0.01 deg; joints [24.718, -40.074, 95.743, -151.043, 59.784, 165.534]
  MoveL 9318 to (-392.35, -27.6, -49.62) mm, rotated rx 180 ry 0 rz 0.01 deg; joints [24.91, -40.248, 96.136, -150.891, 60.027, 165.547]
  MoveL 9319 to (-392.91, -21.02, -49.87) mm, rotated rx 180 ry 0 rz 0.01 deg; joints [25.118, -40.089, 95.807, -150.613, 59.936, 165.334]
  MoveL 9320 to (-399.16, -18.89, -50.11) mm, rotated rx 180 ry 0 rz 0.01 deg; joints [25.092, -39.772, 95.148, -150.544, 59.63, 165.154]
  MoveL 9321 to (-403.61, -23.76, -50.35) mm, rotated rx -180 ry 0 rz 0.01 deg; joints [24.865, -39.662, 94.946, -150.77, 59.487, 165.232]
  MoveL 9322 to (-400.95, -29.79, -50.6) mm, rotated rx 180 ry 0 rz 0.01 deg; joints [24.708, -39.877, 95.442, -151.025, 59.689, 165.481]
  MoveL 9323 to (-394.35, -29.77, -50.84) mm, rotated rx 180 ry 0 rz 0.01 deg; joints [24.809, -40.144, 96.039, -151.006, 60.005, 165.608]
  MoveL 9324 to (-391.72, -23.72, -51.09) mm, rotated rx -180 ry 0 rz 0.01 deg; joints [25.048, -40.13, 96.022, -150.739, 60.068, 165.471]
  MoveL 9325 to (-396.2, -18.88, -51.33) mm, rotated rx 180 ry 0 rz 0.01 deg; joints [25.138, -39.838, 95.409, -150.548, 59.814, 165.239]
  MoveL 9326 to (-402.44, -21.05, -51.57) mm, rotated rx -180 ry 0 rz 0.01 deg; joints [24.972, -39.602, 94.932, -150.664, 59.557, 165.197]
  MoveL 9327 to (-402.95, -27.63, -51.82) mm, rotated rx 180 ry 0 rz 0.01 deg; joints [24.749, -39.692, 95.161, -150.952, 59.617, 165.404]
  MoveL 9328 to (-397.13, -30.74, -52.06) mm, rotated rx -180 ry 0 rz 0.01 deg; joints [24.735, -39.984, 95.82, -151.071, 59.933, 165.617]
  MoveL 9329 to (-391.95, -26.66, -52.3) mm, rotated rx 180 ry 0 rz 0.01 deg; joints [24.949, -40.115, 96.117, -150.88, 60.137, 165.589]
  MoveL 9330 to (-393.6, -20.27, -52.55) mm, rotated rx 180 ry 0 rz 0.01 deg; joints [25.133, -39.914, 95.697, -150.614, 59.996, 165.362]
  MoveL 9331 to (-400.12, -19.23, -52.79) mm, rotated rx 180 ry 0 rz 0.01 deg; joints [25.068, -39.606, 95.059, -150.592, 59.69, 165.211]
  MoveL 9332 to (-403.69, -24.78, -53.04) mm, rotated rx -180 ry 0 rz 0.01 deg; joints [24.832, -39.547, 94.966, -150.845, 59.596, 165.328]
  MoveL 9333 to (-400.05, -30.28, -53.28) mm, rotated rx 180 ry 0 rz 0.01 deg; joints [24.707, -39.792, 95.528, -151.074, 59.838, 165.577]
  MoveL 9334 to (-393.54, -29.14, -53.52) mm, rotated rx -180 ry 0 rz 0.01 deg; joints [24.844, -40.034, 96.069, -151.006, 60.138, 165.667]
  MoveL 9335 to (-391.97, -22.73, -53.77) mm, rotated rx 180 ry 0 rz 0.01 deg; joints [25.078, -39.968, 95.941, -150.728, 60.146, 165.5]
  MoveL 9336 to (-397.21, -18.72, -54.01) mm, rotated rx 180 ry 0 rz 0.01 deg; joints [25.13, -39.66, 95.294, -150.576, 59.866, 165.279]
  MoveL 9337 to (-402.99, -21.91, -54.26) mm, rotated rx -180 ry 0 rz 0.01 deg; joints [24.937, -39.463, 94.901, -150.734, 59.642, 165.278]
  MoveL 9338 to (-402.39, -28.48, -54.5) mm, rotated rx 180 ry 0 rz 0.01 deg; joints [24.732, -39.6, 95.232, -151.018, 59.754, 165.505]
  MoveC 9339 to (-398.64, -30.57, -54.5) mm, rotated rx -180 ry 0 rz 0.01 deg; joints [24.72, -39.797, 95.66, -151.096, 59.954, 165.641] to (-394.51, -29.39, -54.5) mm, rotated rx -180 ry 0 rz 0.01 deg; joints [24.821, -39.949, 95.986, -151.032, 60.132, 165.681]
  MoveC 9340 to (-392.43, -25.64, -54.5) mm, rotated rx 180 ry 0 rz 0.01 deg; joints [24.976, -39.967, 96.017, -150.863, 60.186, 165.601] to (-393.6, -21.52, -54.5) mm, rotated rx 180 ry 0 rz 0.01 deg; joints [25.094, -39.841, 95.737, -150.69, 60.084, 165.448]
  MoveL 9341 to (-395.34, -19.33, -54.5) mm, rotated rx -180 ry 0 rz 0.01 deg; joints [25.139, -39.726, 95.487, -150.602, 59.979, 165.346]
  MoveC 9342 to (-397.17, -18.8, -54.5) mm, rotated rx -180 ry 0 rz 0.01 deg; joints [25.128, -39.639, 95.298, -150.585, 59.887, 165.295] to (-398.28, -20.35, -54.5) mm, rotated rx -180 ry 0 rz 0.01 deg; joints [25.06, -39.622, 95.264, -150.655, 59.854, 165.323]
  MoveL 9343 to (-398.28, -23.65, -54.5) mm, rotated rx 180 ry 0 rz 0.01 deg; joints [24.952, -39.684, 95.403, -150.797, 59.891, 165.429]
  MoveC 9344 to (-397.66, -25.15, -54.5) mm, rotated rx -180 ry 0 rz 0.01 deg; joints [24.913, -39.738, 95.523, -150.859, 59.937, 165.488] to (-396.16, -25.76, -54.5) mm, rotated rx 180 ry 0 rz 0.01 deg; joints [24.915, -39.812, 95.684, -150.881, 60.014, 165.535]
  MoveL 9345 to (-394.29, -25.76, -54.5) mm, rotated rx -180 ry 0 rz 0.01 deg; joints [24.944, -39.891, 95.854, -150.875, 60.101, 165.57]
  MoveC 9346 to (-392.53, -24.66, -54.5) mm, rotated rx -180 ry 0 rz 0.01 deg; joints [25.007, -39.945, 95.967, -150.821, 60.171, 165.568] to (-392.76, -22.59, -54.5) mm, rotated rx -180 ry 0 rz 0.01 deg; joints [25.072, -39.896, 95.859, -150.733, 60.136, 165.498]
  MoveL 9347 to (-393.6, -21.52, -54.5) mm, rotated rx -180 ry 0 rz 0.01 deg; joints [25.094, -39.841, 95.737, -150.69, 60.084, 165.448]
  MoveL 9348 to (-394.1, -21.14, -54.33) mm, rotated rx 180 ry 0 rz 0.01 deg; joints [25.098, -39.821, 95.677, -150.673, 60.05, 165.423]
  MoveL 9349 to (-394.55, -21.04, -53.87) mm, rotated rx -180 ry 0 rz 0.01 deg; joints [25.094, -39.823, 95.635, -150.665, 60.011, 165.4]
  MoveL 9350 to (-394.72, -21.04, -53.23) mm, rotated rx -180 ry 0 rz 0.01 deg; joints [25.091, -39.847, 95.623, -150.659, 59.979, 165.382]
  Set speed (1000.0 mm/s)
  MoveL 9351 to (-394.72, -21.04, 11) mm, rotated rx -180 ry 0 rz 0.01 deg; joints [25.051, -42.942, 95.855, -149.84, 57.481, 163.743]
  Set speed (1000.0 mm/s)
  MoveL 9352 to (-396.5, -24.43, 11) mm, rotated rx 180 ry 0 rz 0.01 deg; joints [24.913, -42.93, 95.837, -149.995, 57.434, 163.825]
  Set speed (100.0 mm/s)
  MoveL 9353 to (-396.5, -24.43, -33.5) mm, rotated rx -180 ry 0 rz 0.01 deg; joints [24.941, -40.802, 95.712, -150.577, 59.182, 164.975]
  MoveL 9354 to (-396.5, -24.43, -53.23) mm, rotated rx -180 ry 0 rz 0.01 deg; joints [24.953, -39.836, 95.605, -150.81, 59.935, 165.456]
  MoveL 9355 to (-397.2, -25.49, -54.5) mm, rotated rx 180 ry 0 rz 0.01 deg; joints [24.908, -39.763, 95.578, -150.873, 59.963, 165.507]
  MoveL 9356 to (-400.74, -30.86, -54.5) mm, rotated rx 180 ry 0 rz 0.01 deg; joints [24.678, -39.714, 95.481, -151.115, 59.859, 165.611]
  MoveL 9357 to (-399.88, -31.14, -54.5) mm, rotated rx -180 ry 0 rz 0.01 deg; joints [24.682, -39.755, 95.571, -151.124, 59.902, 165.636]
  MoveL 9358 to (-398.96, -31.27, -54.5) mm, rotated rx -180 ry 0 rz 0.01 deg; joints [24.692, -39.796, 95.66, -151.127, 59.946, 165.657]
  MoveL 9359 to (-367.82, -31.27, -54.5) mm, rotated rx 180 ry 0 rz 0.01 deg; joints [25.171, -41.09, 98.449, -151.004, 61.383, 166.223]
  MoveL 9360 to (-374.18, -29.32, -54.5) mm, rotated rx 180 ry 0 rz 0.01 deg; joints [25.137, -40.794, 97.806, -150.949, 61.07, 166.049]
  MoveL 9361 to (-374.68, -29.13, -54.5) mm, rotated rx 180 ry 0 rz 0.01 deg; joints [25.135, -40.77, 97.754, -150.943, 61.045, 166.034]
  MoveL 9362 to (-375.84, -28.56, -54.5) mm, rotated rx -180 ry 0 rz 0.01 deg; joints [25.136, -40.711, 97.627, -150.924, 60.985, 165.996]
  MoveL 9363 to (-376.27, -28.32, -54.5) mm, rotated rx -180 ry 0 rz 0.01 deg; joints [25.137, -40.689, 97.579, -150.915, 60.963, 165.98]
  MoveL 9364 to (-386.1, -21.63, -54.5) mm, rotated rx -180 ry 0 rz 0.01 deg; joints [25.206, -40.157, 96.419, -150.668, 60.433, 165.591]
  MoveL 9365 to (-386.52, -21.3, -54.5) mm, rotated rx 180 ry 0 rz 0.01 deg; joints [25.21, -40.134, 96.367, -150.655, 60.41, 165.573]
  MoveL 9366 to (-387.27, -20.6, -54.5) mm, rotated rx 180 ry 0 rz 0.01 deg; joints [25.222, -40.089, 96.271, -150.628, 60.368, 165.537]
  MoveL 9367 to (-387.6, -20.24, -54.5) mm, rotated rx -180 ry 0 rz 0.01 deg; joints [25.228, -40.069, 96.225, -150.614, 60.348, 165.52]
  MoveL 9368 to (-395.31, -10.51, -54.5) mm, rotated rx -180 ry 0 rz 0.01 deg; joints [25.427, -39.56, 95.112, -150.222, 59.878, 165.064]
  MoveL 9369 to (-395.6, -10.08, -54.5) mm, rotated rx 180 ry 0 rz 0.01 deg; joints [25.436, -39.54, 95.068, -150.205, 59.86, 165.045]
  MoveL 9370 to (-399.67, -2.97, -54.5) mm, rotated rx 180 ry 0 rz 0.01 deg; joints [25.604, -39.229, 94.389, -149.911, 59.587, 164.736]
  MoveL 9371 to (-399.88, -2.52, -54.5) mm, rotated rx 180 ry 0 rz 0.01 deg; joints [25.616, -39.211, 94.35, -149.892, 59.572, 164.717]
  MoveL 9372 to (-403.78, 7.43, -54.5) mm, rotated rx 180 ry 0 rz 0.01 deg; joints [25.876, -38.849, 93.554, -149.473, 59.274, 164.313]
  MoveL 9373 to (-403.78, -26.41, -54.5) mm, rotated rx 180 ry 0 rz 0.01 deg; joints [24.778, -39.502, 95.018, -150.933, 59.666, 165.413]
  MoveL 9374 to (-403.58, -27.62, -54.5) mm, rotated rx 180 ry 0 rz 0.01 deg; joints [24.742, -39.533, 95.087, -150.984, 59.689, 165.455]
  MoveL 9375 to (-403.27, -28.44, -54.5) mm, rotated rx 180 ry 0 rz 0.01 deg; joints [24.72, -39.561, 95.149, -151.019, 59.713, 165.487]
  MoveL 9376 to (-403.17, -28.62, -54.5) mm, rotated rx -180 ry 0 rz 0.01 deg; joints [24.715, -39.569, 95.167, -151.026, 59.72, 165.495]
  MoveL 9377 to (-402.57, -28.71, -54.5) mm, rotated rx -180 ry 0 rz 0.01 deg; joints [24.722, -39.596, 95.225, -151.028, 59.749, 165.509]
  MoveL 9378 to (-401.12, -27.44, -54.5) mm, rotated rx 180 ry 0 rz 0.01 deg; joints [24.785, -39.634, 95.304, -150.969, 59.802, 165.496]
  MoveL 9379 to (-394.76, -24.03, -54.5) mm, rotated rx -180 ry 0 rz 0.01 deg; joints [24.994, -39.839, 95.739, -150.802, 60.06, 165.507]
  MoveL 9380 to (-392.32, -23.48, -54.5) mm, rotated rx 180 ry 0 rz 0.01 deg; joints [25.049, -39.931, 95.936, -150.77, 60.166, 165.534]
  MoveL 9381 to (-391.95, -22.82, -54.5) mm, rotated rx -180 ry 0 rz 0.01 deg; joints [25.077, -39.935, 95.942, -150.74, 60.176, 165.52]
  MoveL 9382 to (-397.13, -18.73, -54.74) mm, rotated rx 180 ry 0 rz 0.01 deg; joints [25.131, -39.627, 95.298, -150.584, 59.898, 165.299]
  MoveL 9383 to (-402.95, -21.83, -54.99) mm, rotated rx 180 ry 0 rz 0.01 deg; joints [24.941, -39.427, 94.897, -150.739, 59.67, 165.294]
  MoveL 9384 to (-402.45, -28.41, -55.23) mm, rotated rx 180 ry 0 rz 0.01 deg; joints [24.733, -39.56, 95.219, -151.023, 59.779, 165.519]
  MoveL 9385 to (-396.22, -30.59, -55.48) mm, rotated rx -180 ry 0 rz 0.01 deg; joints [24.756, -39.851, 95.875, -151.1, 60.104, 165.71]
  MoveL 9386 to (-391.72, -25.76, -55.72) mm, rotated rx 180 ry 0 rz 0.01 deg; joints [24.984, -39.939, 96.078, -150.88, 60.267, 165.647]
  MoveL 9387 to (-394.34, -19.7, -55.96) mm, rotated rx -180 ry 0 rz 0.01 deg; joints [25.143, -39.703, 95.584, -150.631, 60.084, 165.412]
  MoveL 9388 to (-400.94, -19.67, -56.21) mm, rotated rx -180 ry 0 rz 0.01 deg; joints [25.043, -39.412, 94.981, -150.654, 59.785, 165.292]
  MoveL 9389 to (-403.62, -25.71, -56.45) mm, rotated rx -180 ry 0 rz 0.01 deg; joints [24.805, -39.399, 94.99, -150.924, 59.738, 165.44]
  MoveL 9390 to (-399.17, -30.58, -56.7) mm, rotated rx -180 ry 0 rz 0.01 deg; joints [24.713, -39.666, 95.599, -151.123, 60.012, 165.684]
  MoveL 9391 to (-392.92, -28.46, -56.94) mm, rotated rx 180 ry 0 rz 0.01 deg; joints [24.878, -39.878, 96.075, -151.013, 60.289, 165.739]
  MoveL 9392 to (-392.35, -21.88, -57.18) mm, rotated rx 180 ry 0 rz 0.01 deg; joints [25.103, -39.767, 95.849, -150.732, 60.248, 165.547]
  MoveL 9393 to (-398.15, -18.72, -57.43) mm, rotated rx -180 ry 0 rz 0.01 deg; joints [25.117, -39.452, 95.187, -150.618, 59.951, 165.344]
  MoveL 9394 to (-403.37, -22.77, -57.67) mm, rotated rx 180 ry 0 rz 0.01 deg; joints [24.906, -39.295, 94.881, -150.811, 59.762, 165.38]
  MoveL 9395 to (-401.76, -29.17, -57.91) mm, rotated rx 180 ry 0 rz 0.01 deg; joints [24.721, -39.47, 95.296, -151.084, 59.921, 165.619]
  MoveL 9396 to (-395.25, -30.26, -58.16) mm, rotated rx 180 ry 0 rz 0.01 deg; joints [24.784, -39.753, 95.932, -151.113, 60.247, 165.781]
  MoveL 9397 to (-391.63, -24.74, -58.4) mm, rotated rx -180 ry 0 rz 0.01 deg; joints [25.021, -39.79, 96.026, -150.866, 60.361, 165.68]
  MoveL 9398 to (-395.24, -19.21, -58.65) mm, rotated rx 180 ry 0 rz 0.01 deg; joints [25.147, -39.523, 95.464, -150.644, 60.138, 165.444]
  MoveL 9399 to (-401.75, -20.3, -58.89) mm, rotated rx 180 ry 0 rz 0.01 deg; joints [25.012, -39.257, 94.916, -150.714, 59.855, 165.361]
  MoveL 9400 to (-403.37, -26.7, -59.13) mm, rotated rx -180 ry 0 rz 0.01 deg; joints [24.778, -39.296, 95.037, -150.997, 59.862, 165.539]
  MoveL 9401 to (-398.16, -30.75, -59.38) mm, rotated rx 180 ry 0 rz 0.01 deg; joints [24.724, -39.579, 95.68, -151.157, 60.163, 165.771]
  MoveL 9402 to (-392.36, -27.6, -59.62) mm, rotated rx 180 ry 0 rz 0.01 deg; joints [24.916, -39.752, 96.072, -151.005, 60.406, 165.786]
  MoveL 9403 to (-392.91, -21.03, -59.87) mm, rotated rx 180 ry 0 rz 0.01 deg; joints [25.124, -39.595, 95.744, -150.727, 60.313, 165.574]
  MoveL 9404 to (-399.16, -18.89, -60.11) mm, rotated rx 180 ry 0 rz 0.01 deg; joints [25.098, -39.28, 95.085, -150.659, 60.006, 165.394]
  MoveL 9405 to (-403.62, -23.76, -60.35) mm, rotated rx 180 ry 0 rz 0.01 deg; joints [24.871, -39.171, 94.882, -150.885, 59.862, 165.47]
  MoveL 9406 to (-400.95, -29.79, -60.6) mm, rotated rx -180 ry 0 rz 0.01 deg; joints [24.714, -39.383, 95.378, -151.139, 60.067, 165.717]
  MoveL 9407 to (-394.35, -29.78, -60.84) mm, rotated rx 180 ry 0 rz 0.01 deg; joints [24.815, -39.648, 95.975, -151.119, 60.385, 165.846]
  MoveL 9408 to (-391.72, -23.73, -61.09) mm, rotated rx -180 ry 0 rz 0.01 deg; joints [25.054, -39.634, 95.958, -150.853, 60.446, 165.71]
  MoveL 9409 to (-396.21, -18.88, -61.33) mm, rotated rx -180 ry 0 rz 0.01 deg; joints [25.144, -39.344, 95.345, -150.663, 60.189, 165.479]
  MoveL 9410 to (-402.44, -21.05, -61.57) mm, rotated rx 180 ry 0 rz 0.01 deg; joints [24.978, -39.11, 94.867, -150.779, 59.931, 165.435]
  MoveL 9411 to (-402.96, -27.63, -61.82) mm, rotated rx -180 ry 0 rz 0.01 deg; joints [24.756, -39.198, 95.096, -151.066, 59.993, 165.64]
  MoveL 9412 to (-397.14, -30.75, -62.06) mm, rotated rx -180 ry 0 rz 0.01 deg; joints [24.741, -39.489, 95.754, -151.183, 60.311, 165.853]
  MoveL 9413 to (-391.95, -26.67, -62.3) mm, rotated rx 180 ry 0 rz 0.01 deg; joints [24.955, -39.618, 96.052, -150.993, 60.516, 165.827]
  MoveL 9414 to (-393.6, -20.28, -62.55) mm, rotated rx 180 ry 0 rz 0.01 deg; joints [25.139, -39.418, 95.631, -150.728, 60.373, 165.601]
  MoveL 9415 to (-400.12, -19.23, -62.79) mm, rotated rx 180 ry 0 rz 0.01 deg; joints [25.074, -39.113, 94.993, -150.707, 60.064, 165.45]
  MoveL 9416 to (-403.7, -24.77, -63.04) mm, rotated rx 180 ry 0 rz 0.01 deg; joints [24.839, -39.054, 94.899, -150.959, 59.97, 165.564]
  MoveL 9417 to (-400.05, -30.28, -63.28) mm, rotated rx 180 ry 0 rz 0.01 deg; joints [24.714, -39.297, 95.461, -151.186, 60.215, 165.812]
  MoveL 9418 to (-393.55, -29.15, -63.52) mm, rotated rx 180 ry 0 rz 0.01 deg; joints [24.85, -39.537, 96.002, -151.118, 60.516, 165.904]
  MoveL 9419 to (-391.97, -22.74, -63.77) mm, rotated rx 180 ry 0 rz 0.01 deg; joints [25.085, -39.472, 95.874, -150.841, 60.523, 165.738]
  MoveL 9420 to (-397.21, -18.72, -64.01) mm, rotated rx 180 ry 0 rz 0.01 deg; joints [25.136, -39.165, 95.227, -150.69, 60.24, 165.518]
  MoveL 9421 to (-402.99, -21.91, -64.26) mm, rotated rx -180 ry 0 rz 0.01 deg; joints [24.944, -38.97, 94.834, -150.847, 60.015, 165.515]
  MoveL 9422 to (-402.4, -28.48, -64.5) mm, rotated rx 180 ry 0 rz 0.01 deg; joints [24.738, -39.105, 95.164, -151.13, 60.13, 165.74]
  MoveC 9423 to (-394.52, -29.4, -64.5) mm, rotated rx -180 ry 0 rz 0.01 deg; joints [24.827, -39.452, 95.918, -151.143, 60.51, 165.916] to (-393.61, -21.52, -64.5) mm, rotated rx -180 ry 0 rz 0.01 deg; joints [25.1, -39.345, 95.67, -150.803, 60.46, 165.686]
  MoveL 9424 to (-395.34, -19.33, -64.5) mm, rotated rx -180 ry 0 rz 0.01 deg; joints [25.145, -39.231, 95.42, -150.715, 60.353, 165.584]
  MoveC 9425 to (-397.17, -18.8, -64.5) mm, rotated rx -180 ry 0 rz 0.01 deg; joints [25.134, -39.144, 95.231, -150.698, 60.261, 165.533] to (-398.28, -20.35, -64.5) mm, rotated rx -180 ry 0 rz 0.01 deg; joints [25.066, -39.127, 95.196, -150.769, 60.228, 165.561]
  MoveL 9426 to (-398.28, -23.65, -64.5) mm, rotated rx 180 ry 0 rz 0.01 deg; joints [24.959, -39.189, 95.336, -150.91, 60.267, 165.665]
  MoveC 9427 to (-397.66, -25.15, -64.5) mm, rotated rx 180 ry 0 rz 0.01 deg; joints [24.919, -39.242, 95.455, -150.972, 60.313, 165.724] to (-396.16, -25.77, -64.5) mm, rotated rx 180 ry 0 rz 0.01 deg; joints [24.921, -39.316, 95.617, -150.993, 60.391, 165.772]
  MoveL 9428 to (-394.3, -25.77, -64.5) mm, rotated rx -180 ry 0 rz 0.01 deg; joints [24.95, -39.394, 95.786, -150.987, 60.478, 165.807]
  MoveC 9429 to (-392.53, -24.66, -64.5) mm, rotated rx 180 ry 0 rz 0.01 deg; joints [25.013, -39.448, 95.899, -150.933, 60.547, 165.805] to (-392.76, -22.59, -64.5) mm, rotated rx -180 ry 0 rz 0.01 deg; joints [25.078, -39.4, 95.792, -150.846, 60.512, 165.736]
  MoveL 9430 to (-393.61, -21.52, -64.5) mm, rotated rx 180 ry 0 rz 0.01 deg; joints [25.1, -39.345, 95.67, -150.803, 60.46, 165.686]
  MoveC 9431 to (-394.38, -21.14, -64.5) mm, rotated rx 180 ry 0 rz 0.01 deg; joints [25.1, -39.305, 95.584, -150.789, 60.42, 165.66] to (-395.16, -21.5, -64.5) mm, rotated rx -180 ry 0 rz 0.01 deg; joints [25.077, -39.279, 95.528, -150.807, 60.387, 165.656]
  MoveL 9432 to (-401.47, -29.1, -64.5) mm, rotated rx -180 ry 0 rz 0.01 deg; joints [24.731, -39.155, 95.274, -151.154, 60.18, 165.777]
  MoveL 9433 to (-401.19, -30.62, -64.5) mm, rotated rx -180 ry 0 rz 0.01 deg; joints [24.686, -39.195, 95.364, -151.218, 60.212, 165.83]
  MoveL 9434 to (-400.74, -30.86, -64.5) mm, rotated rx -180 ry 0 rz 0.01 deg; joints [24.685, -39.218, 95.414, -151.227, 60.235, 165.846]
  MoveL 9435 to (-399.88, -31.14, -64.5) mm, rotated rx -180 ry 0 rz 0.01 deg; joints [24.689, -39.259, 95.504, -151.236, 60.279, 165.871]
  MoveL 9436 to (-398.96, -31.27, -64.5) mm, rotated rx 180 ry 0 rz 0.01 deg; joints [24.698, -39.3, 95.593, -151.239, 60.324, 165.892]
  MoveL 9437 to (-367.91, -31.27, -64.5) mm, rotated rx 180 ry 0 rz 0.01 deg; joints [25.176, -40.58, 98.375, -151.112, 61.765, 166.46]
  MoveL 9438 to (-374.2, -29.32, -64.5) mm, rotated rx -180 ry 0 rz 0.01 deg; joints [25.143, -40.289, 97.737, -151.058, 61.453, 166.287]
  MoveL 9439 to (-374.74, -29.1, -64.5) mm, rotated rx 180 ry 0 rz 0.01 deg; joints [25.142, -40.263, 97.68, -151.051, 61.426, 166.27]
  MoveL 9440 to (-376.35, -28.27, -64.5) mm, rotated rx -180 ry 0 rz 0.01 deg; joints [25.144, -40.182, 97.502, -151.023, 61.342, 166.216]
  MoveL 9441 to (-376.73, -28.05, -64.5) mm, rotated rx 180 ry 0 rz 0.01 deg; joints [25.146, -40.163, 97.46, -151.015, 61.322, 166.202]
  MoveL 9442 to (-386.38, -21.4, -64.5) mm, rotated rx -180 ry 0 rz 0.01 deg; joints [25.215, -39.643, 96.317, -150.771, 60.796, 165.818]
  MoveL 9443 to (-386.79, -21.06, -64.5) mm, rotated rx 180 ry 0 rz 0.01 deg; joints [25.22, -39.62, 96.266, -150.758, 60.773, 165.8]
  MoveL 9444 to (-387.29, -20.58, -64.5) mm, rotated rx -180 ry 0 rz 0.01 deg; joints [25.228, -39.59, 96.201, -150.74, 60.744, 165.775]
  MoveL 9445 to (-387.61, -20.23, -64.5) mm, rotated rx 180 ry 0 rz 0.01 deg; joints [25.234, -39.57, 96.157, -150.726, 60.725, 165.758]
  MoveL 9446 to (-395.31, -10.5, -64.5) mm, rotated rx 180 ry 0 rz 0.01 deg; joints [25.433, -39.066, 95.045, -150.337, 60.25, 165.304]
  MoveL 9447 to (-395.6, -10.08, -64.5) mm, rotated rx 180 ry 0 rz 0.01 deg; joints [25.443, -39.046, 95.001, -150.32, 60.232, 165.285]
  MoveL 9448 to (-399.67, -2.97, -64.5) mm, rotated rx -180 ry 0 rz 0.01 deg; joints [25.611, -38.738, 94.321, -150.028, 59.956, 164.978]
  MoveL 9449 to (-399.88, -2.53, -64.5) mm, rotated rx 180 ry 0 rz 0.01 deg; joints [25.621, -38.721, 94.283, -150.009, 59.941, 164.959]
  MoveL 9450 to (-403.78, 7.36, -64.5) mm, rotated rx -180 ry 0 rz 0.01 deg; joints [25.88, -38.362, 93.49, -149.596, 59.639, 164.559]
  MoveL 9451 to (-403.78, -26.41, -64.5) mm, rotated rx -180 ry 0 rz 0.01 deg; joints [24.785, -39.008, 94.951, -151.046, 60.04, 165.649]
  MoveL 9452 to (-403.58, -27.62, -64.5) mm, rotated rx 180 ry 0 rz 0.01 deg; joints [24.748, -39.039, 95.019, -151.097, 60.064, 165.691]
  MoveL 9453 to (-403.27, -28.44, -64.5) mm, rotated rx 180 ry 0 rz 0.01 deg; joints [24.726, -39.067, 95.082, -151.131, 60.088, 165.722]
  MoveL 9454 to (-403.17, -28.62, -64.5) mm, rotated rx 180 ry 0 rz 0.01 deg; joints [24.722, -39.075, 95.099, -151.139, 60.095, 165.73]
  MoveL 9455 to (-402.71, -29.05, -64.33) mm, rotated rx 180 ry 0 rz 0.01 deg; joints [24.714, -39.111, 95.16, -151.154, 60.115, 165.748]
  MoveL 9456 to (-402.28, -29.2, -63.87) mm, rotated rx 180 ry 0 rz 0.01 deg; joints [24.716, -39.155, 95.21, -151.154, 60.12, 165.75]
  MoveL 9457 to (-402.11, -29.22, -63.23) mm, rotated rx -180 ry 0 rz 0.01 deg; joints [24.717, -39.194, 95.23, -151.147, 60.104, 165.739]
  Set speed (1000.0 mm/s)
  MoveL 9458 to (-402.11, -29.22, 15) mm, rotated rx -180 ry 0 rz 0.01 deg; joints [24.668, -42.962, 95.531, -150.164, 57.068, 163.778]
  Set speed (1000.0 mm/s)
  MoveL 9459 to (-402.11, -29.22, 15) mm, rotated rx -180 ry 0 rz 0.01 deg; joints [24.668, -42.962, 95.531, -150.164, 57.068, 163.778]
